// TwinCAT 3 PLC project STANDARD
// ProgramVersion: 3.1.4023.0
// libraries:
//   Tc2_Standard, * (Beckhoff Automation GmbH)
//   Tc2_System, * (Beckhoff Automation GmbH)
//   Tc3_Module, * (Beckhoff Automation GmbH)
// project tree:
//   / MAIN.TcPOU, PlcTask.TcTTO
//   TC3Sys/process/ IProcess.TcIO (not stored)
//   TC3Sys/utils/ Test.TcPOU (not stored), TestProcess.TcPOU (not stored)
// real-time tasks:
//   TASK PlcTask: cycle T#10ms, priority 20, ADS port 350
// I/O:
//   DEVICE Master1 (EtherCAT), AmsNetId 192.168.7.114.2.1
//     Term 1 (EK1101) [EK1101 EtherCAT Coupler (2A E-Bus, ID switch)]
//       Term 5 (EL1008) [EL1008 8Ch. Dig. Input 24V, 3ms]
//     Term 2 (EK1101) [EK1101 EtherCAT Coupler (2A E-Bus, ID switch)]
//       Term 3 (EL1904) [EL1904, 4 Ch. Safety Input 24V, TwinSAFE]
//         modules: Module 1 (FSOES)
//       Term 4 (EL9011) [EL9011 End Terminal]
// variable links:
//   STANDARD Instance <-> Master1 (EtherCAT)/Term 1 (EK1101)/Term 5 (EL1008)
//     PlcTask Inputs/MAIN.j_digitalInput1 <-> Channel 1/Input

CONFIGURATION STANDARD
    RESOURCE PLC ON TwinCAT3
        TASK PlcTask(INTERVAL := T#10ms, PRIORITY := 20);
        PROGRAM MAIN WITH PlcTask : MAIN;
    END_RESOURCE
END_CONFIGURATION

// ---- MAIN.TcPOU
PROGRAM MAIN
VAR
	j_digitalInput1 AT%I*:BOOL;
	_test:Test;
END_VAR

_test();

END_PROGRAM
